// Mitsubishi GX Works2 project: LRI.gx3   PLC: Q03UDV
// EXERCICIOS

PROGRAM MAIN
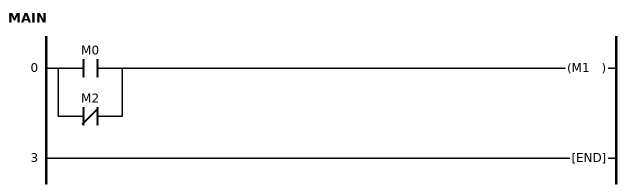
0     LD      M0
      ORI     M2
      OUT     M1
3     END
END_PROGRAM
